TYPE "UDT_CommonStatus"
TITLE = UDT_CommonStatus
VERSION : 0.1
//User-defined structure of common statuses.
   STRUCT
      SafetyStop { ExternalAccessible := 'False'; ExternalVisible := 'False'; ExternalWritable := 'False'} : Bool;   // Emergancy stop
      Error { ExternalAccessible := 'False'; ExternalVisible := 'False'; ExternalWritable := 'False'} : Bool;   // An error is active
      Warning { ExternalAccessible := 'False'; ExternalVisible := 'False'; ExternalWritable := 'False'} : Bool;   // A warning is active
      ManualRun { ExternalAccessible := 'False'; ExternalVisible := 'False'; ExternalWritable := 'False'} : Bool;   // Running in manual mode
      Manual { ExternalAccessible := 'False'; ExternalVisible := 'False'; ExternalWritable := 'False'} : Bool;   // In manual mode
      Halted { ExternalAccessible := 'False'; ExternalVisible := 'False'; ExternalWritable := 'False'} : Bool;   // Halted
      Dieback { ExternalAccessible := 'False'; ExternalVisible := 'False'; ExternalWritable := 'False'} : Bool;   // In dieback
      Stopped { ExternalAccessible := 'False'; ExternalVisible := 'False'; ExternalWritable := 'False'} : Bool;   // Stopped
      Running { ExternalAccessible := 'False'; ExternalVisible := 'False'; ExternalWritable := 'False'} : Bool;   // Running
      EnergySave { ExternalAccessible := 'False'; ExternalVisible := 'False'; ExternalWritable := 'False'} : Bool;   // In energy saving mode
      AutoON { ExternalAccessible := 'False'; ExternalVisible := 'False'; ExternalWritable := 'False'} : Bool;   // Automatic started
   END_STRUCT;

END_TYPE

TYPE "UDT_GINStandard"
VERSION : 0.1
   STRUCT
      Destination : Array[0..20] of DInt;   // Destination
      Identification : Struct   // Barcode identification
         GoodRead { ExternalAccessible := 'False'; ExternalVisible := 'False'; ExternalWritable := 'False'} : Bool;   // Barcode read was succesful
         NoRead { ExternalAccessible := 'False'; ExternalVisible := 'False'; ExternalWritable := 'False'} : Bool;   // Barcode read was unsuccesful
         MultiRead { ExternalAccessible := 'False'; ExternalVisible := 'False'; ExternalWritable := 'False'} : Bool;   // Multiple Barcodes were detected
         Barcode : Array[0..10] of Char;   // Barcode values
      END_STRUCT;
      GinAssigned { ExternalAccessible := 'False'; ExternalVisible := 'False'; ExternalWritable := 'False'} : Bool;   // GIN is assigned to package
      Lost { ExternalAccessible := 'False'; ExternalVisible := 'False'; ExternalWritable := 'False'} : Bool;   // Lost in tracking
      Length : Int;   // Length in mm
      Width : Int;   // Width in mm
      Height : Int;   // Height in mm
      Weight : DInt;   // Weight in g
      PkgTooLong { ExternalAccessible := 'False'; ExternalVisible := 'False'; ExternalWritable := 'False'} : Bool;   // Package is too long
      PkgTooSmall { ExternalAccessible := 'False'; ExternalVisible := 'False'; ExternalWritable := 'False'} : Bool;   // Package is too small
      PkgTooHigh { ExternalAccessible := 'False'; ExternalVisible := 'False'; ExternalWritable := 'False'} : Bool;   // Package is too high
      PkgOverWeight { ExternalAccessible := 'False'; ExternalVisible := 'False'; ExternalWritable := 'False'} : Bool;   // Package is over weight
      TrailingGap : Int;   // Trailing gap size in cm between the package
      LeadingGap : Int;   // Leading gap size in cm between the package
      NrOfRecirculations : Int;   // Number of recirculations
      DestReqSend { ExternalAccessible := 'False'; ExternalVisible := 'False'; ExternalWritable := 'False'} : Bool;   // Destination request sent to high level
      DestRcv { ExternalAccessible := 'False'; ExternalVisible := 'False'; ExternalWritable := 'False'} : Bool;   // Destination received from high level
      SortStatus : Struct   // Sort status of the package
         DivertDestination : Int;   // Destination to which the package is diverted
         GoodDivert { ExternalAccessible := 'False'; ExternalVisible := 'False'; ExternalWritable := 'False'} : Bool;   // Package diverted
         FailedDivert { ExternalAccessible := 'False'; ExternalVisible := 'False'; ExternalWritable := 'False'} : Bool;   // Package failed to divert
         NoDivert : Bool := TRUE;   // Divert is not activated
         NoDivertCause : Struct   // Cause for no divert
            ChuteJam { ExternalAccessible := 'False'; ExternalVisible := 'False'; ExternalWritable := 'False'} : Bool;   // Chute is jammed
            ChuteFull { ExternalAccessible := 'False'; ExternalVisible := 'False'; ExternalWritable := 'False'} : Bool;   // Chute is full
            NoRTR { ExternalAccessible := 'False'; ExternalVisible := 'False'; ExternalWritable := 'False'} : Bool;   // Downstream conveyor is not ready to receive
            DestDisabled { ExternalAccessible := 'False'; ExternalVisible := 'False'; ExternalWritable := 'False'} : Bool;   // Destination is disabled
            TrayDisabled { ExternalAccessible := 'False'; ExternalVisible := 'False'; ExternalWritable := 'False'} : Bool;   // Tray is disabled
            SorterNotAtSpeed { ExternalAccessible := 'False'; ExternalVisible := 'False'; ExternalWritable := 'False'} : Bool;   // Sorter is not at speed
            LeadingGapError { ExternalAccessible := 'False'; ExternalVisible := 'False'; ExternalWritable := 'False'} : Bool;   // Gap size with downstream parcel is not enough
            TrailingGapError { ExternalAccessible := 'False'; ExternalVisible := 'False'; ExternalWritable := 'False'} : Bool;   // Gap size with upstream parcel is not enough
            PkgTooHigh { ExternalAccessible := 'False'; ExternalVisible := 'False'; ExternalWritable := 'False'} : Bool;   // Package is too high to divert
            PkgTooLong { ExternalAccessible := 'False'; ExternalVisible := 'False'; ExternalWritable := 'False'} : Bool;   // Package is too long to divert
            DestNotReachable { ExternalAccessible := 'False'; ExternalVisible := 'False'; ExternalWritable := 'False'} : Bool;   // Sort destionation is not reachable
            InvalidDest { ExternalAccessible := 'False'; ExternalVisible := 'False'; ExternalWritable := 'False'} : Bool;   // Sort destination is invalid
            DestTooLate { ExternalAccessible := 'False'; ExternalVisible := 'False'; ExternalWritable := 'False'} : Bool;   // Destination too late
            NoDestRcv { ExternalAccessible := 'False'; ExternalVisible := 'False'; ExternalWritable := 'False'} : Bool;   // Destination not received from high level
         END_STRUCT;
      END_STRUCT;
   END_STRUCT;

END_TYPE

TYPE "UDT_GINFedEx"
VERSION : 0.1
   STRUCT
      Timestamp : String[17];   // Local time timestamp
      TimeZoneDesignator : String[5];   // Time zone designator
      PackageEntrancePoint : String[14];   // Entrance point, where LLC starts tracking the parcel.
      PackageEntranceState : String[1];   // Entrance state
      PackageExitPoint : String[14];   // Exit point name, where LLC reports the last known tracking point.
      PackageExitState : String[1];   // Exit point state when LLC reports the last known tracking point.
      PalletType : String[2];   // Pallet code for different type of pallets on the market
      Mask : String[1];   // Flag to indicate that a pallet has been mask.
      CellNumber : String[4];   // Tray/Cell number (for loop sorters) or generated by LLC (on line sorters).
      CellsOccupied : String[1];   // Cells occupied by the piece for loop sorters.
      ImageID : String[6];   // Image ID number created by the ADC system.
      ScanUnitType : String[1];   // Scan unit type
      ADCSystemID : String[15];   // Number assigned by the ADC system
      PackageID : String[15];   // Number assigned by the LLC system
      LLCSystemID : String[15];
      HLCPackageID : String[10];   // Unique number for the specific package during it stays in HLC system.
      HLCResultCode : String[16];   // Result code based on processing of the scan event messages.
      ShipmentID : String[6];   // Consignment id of the parcel.
      WeightStatus : String[1];   // Status to indicate if the parcel/pallet has weight on the system.
      ActualDestination : String[6];   // Location code value that describes the actual disposition of the package.
      Destination1 : String[6];   // Location code value that describes where the package should go (Diverter Number).
      Destination2 : String[6];   // Location code value that describes where the package should go (Diverter Number).
      Destination3 : String[6];   // Location code value that describes where the package should go (Diverter Number).
      Destination4 : String[6];   // Location code value that describes where the package should go (Diverter Number).
      Destination5 : String[6];   // Location code value that describes where the package should go (Diverter Number).
      CutOffTimeDestination1 : String[5];   // Cut Off Time in Local Time.
      CutOffTimeDestination2 : String[5];   // Cut Off Time in Local Time.
      CutOffTimeDestination3 : String[5];   // Cut Off Time in Local Time.
      CutOffTimeDestination4 : String[5];   // Cut Off Time in Local Time.
      CutOffTimeDestination5 : String[5];   // Cut Off Time in Local Time.
      ReasonCode1 : String[8];   // Management Code value that describes the result of attempting to route the package to the Destination
      ReasonCode2 : String[8];   // Management Code value that describes the result of attempting to route the package to the Destination
      ReasonCode3 : String[8];   // Management Code value that describes the result of attempting to route the package to the Destination
      ReasonCode4 : String[8];   // Management Code value that describes the result of attempting to route the package to the Destination
      ReasonCode5 : String[8];   // Management Code value that describes the result of attempting to route the package to the Destination
      HLCDataText : String[20];   // Free text for future use.
      Customs : String[1];   // Need to be checked by customs
      DIMSystemID : String[15];   // Identifier of dimensioning system.
      DIMStatus : String[5];   // Basic diagnostic information from the dimensioning system at the moment of the measurement.
      PackageDimLength : String[6];   // Length dimension of package in resolution of dim system.
      PackageDimWidth : String[6];   // Width dimension of package in resolution of dim system.
      PackageDimHeight : String[6];   // Height dimension of package in resolution of dim system.
      DIMUOM : String[2];   // Unit of measure of the package dimensions.
      DimLFTstatusCode : String[8];   // Dimension LFT status code.
      DimConfidence : String[2];   // The level of assurance for the correct dimensions.
      DimensionSource : String[1];   // For combined camera/laser dim acquisition devices. It indicates type of capturing mode
      AlibiDims : String[25];   // Alibi for Dimensions
      SCLSystemID : String[15];   // Identifier of weight scale.
      SCLStatus : String[5];   // Basic diagnostic information from the weight scale system.
      SCLWT : String[6];   // Scale weight of package in resolution of scale system.
      SCLWTUOM : String[2];   // Unit of measurement for Weight
      SCLLFTStatusCode : String[2];   // Scale LFT status code.
      AlibiWeight : String[25];   // Alibi for Weight
      ReasonCode : String[1];   // This code should be used when the SI message has some defect.
      Stackable : String[1];   // If stackable recognition is enabled, Y or N
      Stickerstype : String[2];   // When optical recognition is used to sort
      FlyingDocument : String[1];   // Status to confirm if the document/flyer is prone to fly off the sorter.
      ModeofOperation : String[1];   // Camera Tunnel operational mode format:
      CameraHeadstatus : String[2];   // Diagnostic information on camera/laser heads performing barcode reads.
      PackageDataTruncated : String[1];   // Y = Full length of barcode data exceeds 9999 bytes, data truncated
      TotalBarcodeDataLength : String[4];   // Length of all barcode data that was sent in bytes;
      Barcode1Identification : String[3];   // Barcode identifier code.
      Barcode1status : String[2];   // Barcode confidence factor
      Barcode1datalength : String[4];   // String length of barcode data in bytes; inclusive of this field. Use 0054 as a fixed value
      Barcode1data : String[50];   // Highest priority barcode
      Barcode2Identification : String[3];   // Barcode identifier code.
      Barcode2status : String[2];   // Barcode confidence factor
      Barcode2datalength : String[4];   // String length of barcode data in bytes; inclusive of this field. Use 0054 as a fixed value
      Barcode2data : String[50];   // Highest priority barcode
      Barcode3Identification : String[3];   // Barcode identifier code.
      Barcode3status : String[2];   // Barcode confidence factor
      Barcode3datalength : String[4];   // String length of barcode data in bytes; inclusive of this field. Use 0054 as a fixed value
      Barcode3data : String[50];   // Highest priority barcode
      BarcodeIdentification : String[3];   // Barcode identifier code.
      Barcodestatus : String[2];   // Barcode confidence factor
      Barcodedatalength : String[4];   // String length of barcode data in bytes
      Barcodedata : String[50];   // Sortation barcode
      CustomerID : DInt;   // 6 digits SequentialID (NNNNNN)
      AreaNumber : String[2];   // Package Sequence ID "Area Number"
      PurgeEnabled { ExternalAccessible := 'False'; ExternalVisible := 'False'; ExternalWritable := 'False'} : Bool;   // Purge enabled for parcel: destination overwritten with Purge destination
   END_STRUCT;

END_TYPE

TYPE "UDT_GINUPS"
VERSION : 0.1
   STRUCT
      TRKNUM : String[18];   // Tracking number
      PKGUID : String[32];   // Package ID
      MSGID : String[32];   // Message ID
      Length : Int;   // Camera Length in mm
      Width : Int;   // Camera Width in mm
      Height : Int;   // Camera Height in mm
      Weight : DInt;   // Weight in g
      IDCreated { ExternalAccessible := 'False'; ExternalVisible := 'False'; ExternalWritable := 'False'} : Bool;   // Byte 1, Bit 0 - PLCID created or TrayID Read
      DimDataRcv { ExternalAccessible := 'False'; ExternalVisible := 'False'; ExternalWritable := 'False'} : Bool;   // Byte 1, Bit 1 - Package Dimensional Data Received via Camera Scan Data Message
      PkgWrongInduct { ExternalAccessible := 'False'; ExternalVisible := 'False'; ExternalWritable := 'False'} : Bool;   // Byte 1, Bit 2 - Package Did NOT Induct Properly (Non-Tray Systems)
      IDCalcFromCamID { ExternalAccessible := 'False'; ExternalVisible := 'False'; ExternalWritable := 'False'} : Bool;   // Byte 2, Bit 0 - PLCID/TrayID Calculated From CamID
      UnknownParcelID { ExternalAccessible := 'False'; ExternalVisible := 'False'; ExternalWritable := 'False'} : Bool;   // Byte 2, Bit 4 - Unknown Parcel ID
      UndefinedProblem { ExternalAccessible := 'False'; ExternalVisible := 'False'; ExternalWritable := 'False'} : Bool;   // Byte 2, Bit 5 - Un-Defined Problem
      UnrecognizedCmd { ExternalAccessible := 'False'; ExternalVisible := 'False'; ExternalWritable := 'False'} : Bool;   // Byte 2, Bit 6 - Un-recognized command
      SorterInMainteneceMode { ExternalAccessible := 'False'; ExternalVisible := 'False'; ExternalWritable := 'False'} : Bool;   // Byte 2, Bit 7 - Sorter in Maintenance/Commissioning Mode
      DestUserSusp { ExternalAccessible := 'False'; ExternalVisible := 'False'; ExternalWritable := 'False'} : Bool;   // Byte 3, Bit 3 - Destination User Suspended
      SorterNotSynch { ExternalAccessible := 'False'; ExternalVisible := 'False'; ExternalWritable := 'False'} : Bool;   // Byte 3, Bit 6 - Sorter NOT Synchronized (Tilt Tray Systems)
      PkgDetAtVerCheckPoint { ExternalAccessible := 'False'; ExternalVisible := 'False'; ExternalWritable := 'False'} : Bool;   // Byte 4, Bit 0 - Package Detected at Verification Check Point
      ChuteFullAftrAlterDest { ExternalAccessible := 'False'; ExternalVisible := 'False'; ExternalWritable := 'False'} : Bool;   // Byte 4, Bit 7 - Preferred chute full after passed alternate destination
      ChuteNotAvailAfterAlterDest { ExternalAccessible := 'False'; ExternalVisible := 'False'; ExternalWritable := 'False'} : Bool;   // Byte 5, Bit 0 - Preferred chute not available after passed alternate destination
      PLCRedirected { ExternalAccessible := 'False'; ExternalVisible := 'False'; ExternalWritable := 'False'} : Bool;   // Byte 5, Bit 2 - PLC Redirected
      ThreatParcel { ExternalAccessible := 'False'; ExternalVisible := 'False'; ExternalWritable := 'False'} : Bool;   // Threat parcel
   END_STRUCT;

END_TYPE

TYPE "UDT_GINDHL"
VERSION : 0.1
   STRUCT
      ObjectID : String[10];   // Object ID
      VID : String[16];   // Virtual Item Identifier (VID)
      PieceID : String[40];   // Piece ID barcodes
      SortStrategy : String[1];   // Sort Strategy 1 - Highest priority available , 2 - Nearest
      ParcelReject { ExternalAccessible := 'False'; ExternalVisible := 'False'; ExternalWritable := 'False'} : Bool;   // True - Parcel reject
      Destination : Array[1..6] of Struct   // Destination
         ID : UInt;   // ID
         SortCommandActive { ExternalAccessible := 'False'; ExternalVisible := 'False'; ExternalWritable := 'False'} : Bool;   // Sort command
         ParcelSorted { ExternalAccessible := 'False'; ExternalVisible := 'False'; ExternalWritable := 'False'} : Bool;   // Parcel sorted
         Rejected { ExternalAccessible := 'False'; ExternalVisible := 'False'; ExternalWritable := 'False'} : Bool;   // Parcel rejected
         Reason : Int;   // Reason
      END_STRUCT;
      ParcelLocation : Struct   // Parcel Location
         Current : UInt;   // Current
         Last : UInt;   // Last
         Sort : UInt;   // Sort
      END_STRUCT;
      MFCMessage : Struct   // MFC Sort messages
         Sent : Struct   // Messages sent from the PLC to the MFC system
            SortResult { ExternalAccessible := 'False'; ExternalVisible := 'False'; ExternalWritable := 'False'} : Bool;   // Message Sort Result
            VIDResponse { ExternalAccessible := 'False'; ExternalVisible := 'False'; ExternalWritable := 'False'} : Bool;   // Message VID Response
            ScanReset { ExternalAccessible := 'False'; ExternalVisible := 'False'; ExternalWritable := 'False'} : Bool;   // Message Scan Reset
            XrayResult { ExternalAccessible := 'False'; ExternalVisible := 'False'; ExternalWritable := 'False'} : Bool;   // Message Xray result
            ParcelRegInfo { ExternalAccessible := 'False'; ExternalVisible := 'False'; ExternalWritable := 'False'} : Bool;   // Message Xray registration info
         END_STRUCT;
         Received : Struct   // Messages received from the MFC system to the PLC
            RejectParcel { ExternalAccessible := 'False'; ExternalVisible := 'False'; ExternalWritable := 'False'} : Bool;   // Message Reject Parcel
            Destination { ExternalAccessible := 'False'; ExternalVisible := 'False'; ExternalWritable := 'False'} : Bool;   // Message Destination
            DestinationResent { ExternalAccessible := 'False'; ExternalVisible := 'False'; ExternalWritable := 'False'} : Bool;   // Message Destination Resent
            TemporaryParcelIdentifier { ExternalAccessible := 'False'; ExternalVisible := 'False'; ExternalWritable := 'False'} : Bool;   // Message Temporary Parcel Identifier
            XrayRegistrationInfo { ExternalAccessible := 'False'; ExternalVisible := 'False'; ExternalWritable := 'False'} : Bool;
         END_STRUCT;
      END_STRUCT;
      Xray : Struct   // Xray data structure
         RoutingCode : String[2];   // Routing code
         Group : String[1];   // The group field is used to identify the group of the operator decisions came from in a
         Level : String[1];   // Level field is used to identify which level the operator decision came from in a
         Result : String[1];   // Results can be indicated with the following:A = Accept, R = Reject, U = Unavailable (Timeout), Z = High Threat
         BagIDMessage : Struct   // Message from PLC to Xray
            MessagePrepared { ExternalAccessible := 'False'; ExternalVisible := 'False'; ExternalWritable := 'False'} : Bool;   // The message is prepared and ready to send
            WrongMessageStructure { ExternalAccessible := 'False'; ExternalVisible := 'False'; ExternalWritable := 'False'} : Bool;   // The message has wrong structure
            Sent { ExternalAccessible := 'False'; ExternalVisible := 'False'; ExternalWritable := 'False'} : Bool;   // The message sent by PLC to Xray
            SentTime : String;   // Time when message sent by PLC to Xray
            NotSent { ExternalAccessible := 'False'; ExternalVisible := 'False'; ExternalWritable := 'False'} : Bool;   // The message was not sent from the PLC
            Received { ExternalAccessible := 'False'; ExternalVisible := 'False'; ExternalWritable := 'False'} : Bool;   // The message received by Xray
            TimeReceived : String;   // Time when message received by Xray
            NotReceived { ExternalAccessible := 'False'; ExternalVisible := 'False'; ExternalWritable := 'False'} : Bool;   // The message did not reach Xray
         END_STRUCT;
         DecisionMessage : Struct   // Message from Xray to PLC
            Received { ExternalAccessible := 'False'; ExternalVisible := 'False'; ExternalWritable := 'False'} : Bool;   // The message received by PLC
            ReceivedTime : String;   // The message received by PLC
            NotReceivedOnTime { ExternalAccessible := 'False'; ExternalVisible := 'False'; ExternalWritable := 'False'} : Bool;   // The message did not reach PLC
         END_STRUCT;
      END_STRUCT;
   END_STRUCT;

END_TYPE

TYPE "UDT_GINWCS"
VERSION : 0.1
   STRUCT
      ActionTaken : String;   // Location code value that describes the actual disposition of the package
      Destination1 : String[20];   // Location code value that describes where the package should go (Diverter Number)
      Destination2 : String[20];   // Location code value that describes where the package should go (Diverter Number)
      Destination3 : String[20];   // Location code value that describes where the package should go (Diverter Number)
      Destination4 : String[20];   // Location code value that describes where the package should go (Diverter Number)
      Destination5 : String[20];   // Location code value that describes where the package should go (Diverter Number)
      ReasonCode : String[2];   // Management Code value that describes the result of attempting to route the package to the Destination
      Barcode1 : String;   // Barcode identifier code
      Barcode2 : String;
      Barcode3 : String;
      Barcode4 : String;
   END_STRUCT;

END_TYPE

TYPE "UDT_GINWES"
VERSION : 0.1
   STRUCT
      Barcode : String[40];
   END_STRUCT;

END_TYPE

TYPE "UDT_UPSHealth"
TITLE = UDT_Health
VERSION : 0.1
//User-defined structure of UPS health message data.
   STRUCT
      "Type" : String;
      Failure : DInt;
      Model : String;
      Error : Bool;
   END_STRUCT;

END_TYPE

TYPE "UDT_FifoStatus"
TITLE = UDT_FifoStatus
VERSION : 0.1
//
//User-defined structure of FC_Fifo function status.
//Version History:
//Date              | Version   | Author         | Remark
//24/05/2019  | 0.1           | K.Pokorski   | first release MHSE TIA 15.1
//24/05/2019  | 0.2           | K.Pokorski   | first release MHSE TIA 15.1
//
   STRUCT
      InvalidMode { ExternalAccessible := 'False'; ExternalVisible := 'False'; ExternalWritable := 'False'} : Bool;   // Invalid mode selected
      InvalidMaxNrOfEntries { ExternalAccessible := 'False'; ExternalVisible := 'False'; ExternalWritable := 'False'} : Bool;   // Invalid maximum number of entries or buffer is not an array
      InvalidTotalEntriesStored { ExternalAccessible := 'False'; ExternalVisible := 'False'; ExternalWritable := 'False'} : Bool;   // Invalid total number of entries
      InvalidNextEntryToWrite { ExternalAccessible := 'False'; ExternalVisible := 'False'; ExternalWritable := 'False'} : Bool;   // Invalid number of next entry to write
      InvalidNextEntryToRead { ExternalAccessible := 'False'; ExternalVisible := 'False'; ExternalWritable := 'False'} : Bool;   // Invalid number of next entry to read
      InvalidDataType { ExternalAccessible := 'False'; ExternalVisible := 'False'; ExternalWritable := 'False'} : Bool;   // Message and buffer element data type inconsistent
      FifoPreFull { ExternalAccessible := 'False'; ExternalVisible := 'False'; ExternalWritable := 'False'} : Bool;   // 90 % of FIFO data buffer capacity reached
      FifoFull { ExternalAccessible := 'False'; ExternalVisible := 'False'; ExternalWritable := 'False'} : Bool;   // FIFO data buffer full
   END_STRUCT;

END_TYPE

DATA_BLOCK "DB_Memory"
TITLE = DB_Memory
{ S7_Optimized_Access := 'TRUE' }
AUTHOR : MHSE
VERSION : 3.0
NON_RETAIN
   VAR
      ClockByte { ExternalAccessible := 'False'; ExternalVisible := 'False'; ExternalWritable := 'False'} : Byte;   // System clock byte
      Clock_10Hz { ExternalAccessible := 'False'; ExternalVisible := 'False'; ExternalWritable := 'False'} : Bool;   // 10 Hz system clock bit
      Clock_5Hz { ExternalAccessible := 'False'; ExternalVisible := 'False'; ExternalWritable := 'False'} : Bool;   // 5 Hz system clock bit
      "Clock_2.5Hz" { ExternalAccessible := 'False'; ExternalVisible := 'False'; ExternalWritable := 'False'} : Bool;   // 2.5 Hz system clock bit
      Clock_2Hz { ExternalAccessible := 'False'; ExternalVisible := 'False'; ExternalWritable := 'False'} : Bool;   // 2 Hz system clock bit
      "Clock_1.25Hz" { ExternalAccessible := 'False'; ExternalVisible := 'False'; ExternalWritable := 'False'} : Bool;   // 1.25 Hz system clock bit
      Clock_1Hz { ExternalAccessible := 'False'; ExternalVisible := 'False'; ExternalWritable := 'False'} : Bool;   // 1 Hz system clock bit
      "Clock_0.625Hz" { ExternalAccessible := 'False'; ExternalVisible := 'False'; ExternalWritable := 'False'} : Bool;   // 0.625 Hz system clock bit
      "Clock_0.5Hz" { ExternalAccessible := 'False'; ExternalVisible := 'False'; ExternalWritable := 'False'} : Bool;   // 0.5 Hz system clock bit
      SystemByte { ExternalAccessible := 'False'; ExternalVisible := 'False'; ExternalWritable := 'False'} : Byte;   // System byte
      OSClockByte { ExternalAccessible := 'False'; ExternalVisible := 'False'; ExternalWritable := 'False'} : Byte;   // One shot of clock pulse
      "OS_0.1sec" { ExternalAccessible := 'False'; ExternalVisible := 'False'; ExternalWritable := 'False'} : Bool;   // One shot every 0.1 sec
      "OS_0.2sec" { ExternalAccessible := 'False'; ExternalVisible := 'False'; ExternalWritable := 'False'} : Bool;   // One shot every 0.2 sec
      "OS_0.4sec" { ExternalAccessible := 'False'; ExternalVisible := 'False'; ExternalWritable := 'False'} : Bool;   // One shot every 0.4 sec
      "OS_0.5sec" { ExternalAccessible := 'False'; ExternalVisible := 'False'; ExternalWritable := 'False'} : Bool;   // One shot every 0.5 sec
      "OS_0.8sec" { ExternalAccessible := 'False'; ExternalVisible := 'False'; ExternalWritable := 'False'} : Bool;   // One shot every 0.8 sec
      OS_1sec { ExternalAccessible := 'False'; ExternalVisible := 'False'; ExternalWritable := 'False'} : Bool;   // One shot every 1 sec
      "OS_1.6sec" { ExternalAccessible := 'False'; ExternalVisible := 'False'; ExternalWritable := 'False'} : Bool;   // One shot every 1.6 sec
      OS_2sec { ExternalAccessible := 'False'; ExternalVisible := 'False'; ExternalWritable := 'False'} : Bool;   // One shot every 2 sec
      PrevCycleTime { ExternalAccessible := 'False'; ExternalVisible := 'False'; ExternalWritable := 'False'} : LReal;   // Previous PLC cycle Time
      RuntimeMem { ExternalAccessible := 'False'; ExternalVisible := 'False'; ExternalWritable := 'False'} : LReal;   // Runtime memory
      FirstScan { ExternalAccessible := 'False'; ExternalVisible := 'False'; ExternalWritable := 'False'} : Bool;   // First scan bit
      DiagStatusUpdate { ExternalAccessible := 'False'; ExternalVisible := 'False'; ExternalWritable := 'False'} : Bool;   // Diagnostic status update
      AlwaysTrue { ExternalAccessible := 'False'; ExternalVisible := 'False'; ExternalWritable := 'False'} : Bool;   // Always True bit
      AlwaysFalse { ExternalAccessible := 'False'; ExternalVisible := 'False'; ExternalWritable := 'False'} : Bool;   // Always False bit
      CommissioningFalse { ExternalAccessible := 'False'; ExternalVisible := 'False'; ExternalWritable := 'False'} : Bool;   // Commissioning always false
      CommissioningTrue { ExternalAccessible := 'False'; ExternalVisible := 'False'; ExternalWritable := 'False'} : Bool;   // Commissioning always true
      ReconnectCommand { ExternalAccessible := 'False'; ExternalVisible := 'False'; ExternalWritable := 'False'} : Bool;   // Reconnect command
      ScanMainRack { ExternalAccessible := 'False'; ExternalVisible := 'False'; ExternalWritable := 'False'} : Bool;   // Trigger to check main rack confiuration
      ScanProfinet { ExternalAccessible := 'False'; ExternalVisible := 'False'; ExternalWritable := 'False'} : Bool;   // Scan profinet bit
      Simulation { ExternalAccessible := 'False'; ExternalVisible := 'False'; ExternalWritable := 'False'} : Bool;   // Simulation
      PN1OK { ExternalAccessible := 'False'; ExternalVisible := 'False'; ExternalWritable := 'False'} : Bool;   // Profinet ok
      "Local~PROFINET_IO-System" { ExternalAccessible := 'False'; ExternalVisible := 'False'; ExternalWritable := 'False'} : HW_ANY;   // HW Intentifier of PN-IO System
      "Local~PROFINET_IO-System_1" { ExternalAccessible := 'False'; ExternalVisible := 'False'; ExternalWritable := 'False'} : HW_ANY;   // HW Intentifier of PN-IOSystem 1
      "Local~PROFINET_IO-System_2" { ExternalAccessible := 'False'; ExternalVisible := 'False'; ExternalWritable := 'False'} : HW_ANY;   // HW Intentifier of PN-IOSystem 2
      "Local~PROFINET_IO-System_3" { ExternalAccessible := 'False'; ExternalVisible := 'False'; ExternalWritable := 'False'} : HW_ANY;   // HW Intentifier of PN-IOSystem 3
      "Local~PROFINET_IO-System_4" { ExternalAccessible := 'False'; ExternalVisible := 'False'; ExternalWritable := 'False'} : HW_ANY;   // HW Intentifier of PN-IOSystem 4
      "Local~PROFINET_IO-System_5" { ExternalAccessible := 'False'; ExternalVisible := 'False'; ExternalWritable := 'False'} : HW_ANY;   // HW Intentifier of PN-IOSystem 5
      "Local~PROFINET_IO-System_6" { ExternalAccessible := 'False'; ExternalVisible := 'False'; ExternalWritable := 'False'} : HW_ANY;   // HW Intentifier of PN-IOSystem 6
      "Local~PROFINET_IO-System_7" { ExternalAccessible := 'False'; ExternalVisible := 'False'; ExternalWritable := 'False'} : HW_ANY;   // HW Intentifier of PN-IOSystem 7
      "Local~PROFINET_IO-System_8" { ExternalAccessible := 'False'; ExternalVisible := 'False'; ExternalWritable := 'False'} : HW_ANY;   // HW Intentifier of PN-IOSystem 8
      "Local~PROFINET_IO-System_9" { ExternalAccessible := 'False'; ExternalVisible := 'False'; ExternalWritable := 'False'} : HW_ANY;   // HW Intentifier of PN-IOSystem 9
   END_VAR


BEGIN

END_DATA_BLOCK

TYPE "UDT_GIN"
VERSION : 0.1
   STRUCT
      General { S7_SetPoint := 'False'} : "UDT_GINStandard";
      FedEx { S7_SetPoint := 'False'} : "UDT_GINFedEx";
      UPS { S7_SetPoint := 'False'} : "UDT_GINUPS";
      DHL { S7_SetPoint := 'False'} : "UDT_GINDHL";
      WCS { S7_SetPoint := 'False'} : "UDT_GINWCS";
      WES { S7_SetPoint := 'False'} : "UDT_GINWES";
   END_STRUCT;

END_TYPE

TYPE "UDT_FifoHeader"
TITLE = UDT_FifoHeader
VERSION : 0.1
//User-defined structure of FIFO register header information.
   STRUCT
      Status : Struct   // Status bits
         Empty { ExternalAccessible := 'False'; ExternalVisible := 'False'; ExternalWritable := 'False'} : Bool;   // FIFO Empty
         Prefull { ExternalAccessible := 'False'; ExternalVisible := 'False'; ExternalWritable := 'False'} : Bool;   // FIFO Prefull
         Full { ExternalAccessible := 'False'; ExternalVisible := 'False'; ExternalWritable := 'False'} : Bool;   // FIFO Full
      END_STRUCT;
      NextEntryToRead : Int;   // Next FIFO entry to read
      NextEntryToWrite : Int;   // Next FIFO entry to write
      MaxNrOfEntries : Int;   // Maximum number of FIFO entries
      TotalEntriesStored : Int;   // Total number of FIFO entries
   END_STRUCT;

END_TYPE

TYPE "UDT_EventStatistic"
TITLE = UDT_EventStatistic
VERSION : 0.1
//User-defined structure of event statistic data.
   STRUCT
      NumberOfTimes : DInt;   // Number of times the event occurred since last reset
      LastEventSeconds : DInt;   // Number of seconds of the current or last event
      TotalEventSeconds : DInt;   // Total number of seconds the event occurred since last reset
   END_STRUCT;

END_TYPE

TYPE "UDT_EquipmentControl"
TITLE = UDT_EquipmentControl
VERSION : 0.1
//User-defined structure of equipment control commands.
   STRUCT
      Command : Struct   // Control command
         Start { ExternalAccessible := 'False'; ExternalVisible := 'False'; ExternalWritable := 'False'} : Bool;   // Start conveyor
         Stop { ExternalAccessible := 'False'; ExternalVisible := 'False'; ExternalWritable := 'False'} : Bool;   // Stop conveyor
         Reset { ExternalAccessible := 'False'; ExternalVisible := 'False'; ExternalWritable := 'False'} : Bool;   // Faults reset
         ResetData { ExternalAccessible := 'False'; ExternalVisible := 'False'; ExternalWritable := 'False'} : Bool;   // Statistics reset
         ManualMode { ExternalAccessible := 'False'; ExternalVisible := 'False'; ExternalWritable := 'False'} : Bool;   // Manual mode required
         DisableManualMode { ExternalAccessible := 'False'; ExternalVisible := 'False'; ExternalWritable := 'False'} : Bool;   // Disable manual mode
         AutomaticOn { ExternalAccessible := 'False'; ExternalVisible := 'False'; ExternalWritable := 'False'} : Bool;   // System is started in automatic mode
         StopRequest { ExternalAccessible := 'False'; ExternalVisible := 'False'; ExternalWritable := 'False'} : Bool;
      END_STRUCT;
      Report { S7_SetPoint := 'False'} : "UDT_CommonStatus";   // Conveyors state
      Request : Struct   // Request from equipment
         RestartRequired { ExternalAccessible := 'False'; ExternalVisible := 'False'; ExternalWritable := 'False'} : Bool;   // Restart required from system control
         SignalingRequest { ExternalAccessible := 'False'; ExternalVisible := 'False'; ExternalWritable := 'False'} : Bool;   // Beeper required
         InhibitStop { ExternalAccessible := 'False'; ExternalVisible := 'False'; ExternalWritable := 'False'} : Bool;
      END_STRUCT;
   END_STRUCT;

END_TYPE

FUNCTION "FC_GetNrOfArrayEl" : Int
TITLE = FC_GetNrOfArrayEl
{ S7_Optimized_Access := 'TRUE' }
AUTHOR : MHSE
FAMILY : GeneralSystemFunctions
VERSION : 3.0
// ATTRIBUTES
// AUTO_NUMBER = True
// BLOCK_NUMBER = 19
// END_ATTRIBUTES
//Function to get the number of array elements.
   VAR_INPUT
      iv_Array : Variant;   // Input array
   END_VAR

   VAR_TEMP
      ti_NrOfArrayEl : Int;   // Number of array elements
   END_VAR


BEGIN
	(*
	----------------------------------------------------------------------------------------

	Version history:
	Date        | Version   | Author        | Remark
	----------------------------------------------------------------------------------------
	24/05/2019  | 0.1       | L.Klar        | first release MHS TIA 15.1
	24/07/2019  | 2.0       | L.Klar        | 2.0 MHS library release TIA 15.1
	27/08/2019  | 2.1       | K.Pokorski    | Comments adjusted
	12/11/2019  | 3.0       | P.Majka       | 3.0 MHS library release TIA 15.1
	21/02/2023  | 4.0       | F.Baten       | 4.0 Release TIA 17.5
	*)

	REGION 1 – Number of an array elements

	    IF IS_ARRAY(#iv_Array)                                                  // Input variable is an array
	    THEN

	        #ti_NrOfArrayEl := UDINT_TO_INT(CountOfElements(#iv_Array));

	        // Reset array length if the input variable isn't an array
	    ELSE

	        #ti_NrOfArrayEl := 0;

	    END_IF;

	END_REGION

	REGION 2 – Return output

	    #FC_GetNrOfArrayEl := #ti_NrOfArrayEl;

	END_REGION

END_FUNCTION

TYPE "UDT_UPSScanData2"
TITLE = UDT_ScanData2
VERSION : 0.1
//User-defined structure of UPS SCAN_DATA2 data.
   STRUCT
      MSGID : String;
      CONFLICT_CODE : String;
      BARCODE_ZIP : String;
      BARCODE_TRACK : String;
      BARCODE_PTN : String;
      MAXI_ZIPCODE : String;
      MAXI_COUNTRY : String;
      MAXI_SERVICE : String;
      MAXI_TRACK : String;
      MAXI_SHIPPER : String;
      LENGTH1 : String;
      LENGTH2 : String;
      HEIGHT : String;
      VERTEX : String;
      ORIENTATION : String;
      OVERHANG : String;
      WEIGHT : String;
      APPENDED_DATA : Struct
         Constant_1 : String := '1';
         FRAME_ID : String;
         DIMENSION : String;
         PACKAGE_NUMBER : String;
         BARCODE_1 : String;
         DESCRIPTION_1 : String;
         BARCODE_2 : String;
         DESCRIPTION_2 : String;
         BARCODE_3 : String;
         DESCRIPTION_3 : String;
         Constant_4 : String := '4';
         SCALE_WEIGHT : String;
         Constant_5 : String := '5';
         GIRTH : String;
         Constant_6 : String := '6';
         ERROR_CODE : String;
      END_STRUCT;
   END_STRUCT;

END_TYPE

DATA_BLOCK "DB_GIN"
TITLE = DB_GIN
{ S7_Optimized_Access := 'TRUE' }
AUTHOR : MHSE
FAMILY : GeneralSystemFunctions
VERSION : 3.0
NON_RETAIN
//Data block to store parcels informations.
   VAR
      GIN { ExternalAccessible := 'False'; ExternalVisible := 'False'; ExternalWritable := 'False'; S7_SetPoint := 'False'} : Array[1..1] of "UDT_GIN";   // GIN informations - for project remove unneeded customers and extend array bound range to 9999
   END_VAR


BEGIN

END_DATA_BLOCK

TYPE "UDT_UPSMessage"
VERSION : 0.1
   STRUCT
      SCN { ExternalAccessible := 'False'; ExternalVisible := 'False'; ExternalWritable := 'False'} : String[15];   // Sender Client Name
      SCT { ExternalAccessible := 'False'; ExternalVisible := 'False'; ExternalWritable := 'False'} : String[8];   // Sender Client Type
      RCN { ExternalAccessible := 'False'; ExternalVisible := 'False'; ExternalWritable := 'False'} : String[15];   // Receiver Client Name
      RCT { ExternalAccessible := 'False'; ExternalVisible := 'False'; ExternalWritable := 'False'} : String[8];   // Receiver Client Type
      MT { ExternalAccessible := 'False'; ExternalVisible := 'False'; ExternalWritable := 'False'} : String;   // Message type
      Data { ExternalAccessible := 'False'; ExternalVisible := 'False'; ExternalWritable := 'False'} : Array[1..35] of String[32];   // Buffer for message data fields
   END_STRUCT;

END_TYPE

TYPE "UDT_UPSExternalReader"
VERSION : 0.1
   STRUCT
      NameIdentifier : String := 'CAMERA';   // Device name idetifier
      IPAddress : String[15];
      State : Bool;
      HealthMessage { S7_SetPoint := 'False'} : "UDT_UPSHealth";   // Health message data
      ScanData2Message { S7_SetPoint := 'False'} : "UDT_UPSScanData2";   // ScanData2 message data
   END_STRUCT;

END_TYPE

TYPE "UDT_Connection"
TITLE = UDT_Connection
VERSION : 0.1
//User-defined structure of connection parameters.
   STRUCT
      ActiveEstablished : Bool := FALSE;   // 0 – Passive connection establishment; 1 – Active connection establishment
      Interface_ID : HW_ANY := 64;   // Interface ID of CPU Ethernet interface
      ID : CONN_OUC;   // Unique ID as system reference for the connection
      IP : Array[1..4] of Int;   // IP address
      Port : UInt;   // Port number of the communication partner
      ConTimeout : DInt;   // Maximum waiting time for response from the communication partner [ms]
   END_STRUCT;

END_TYPE

TYPE "UDT_Message"
TITLE = UDT_Message
VERSION : 0.1
//User-defined structure of the message characters array.
   STRUCT
      Character : Array[0..499] of Char;   // Message character
   END_STRUCT;

END_TYPE

TYPE "UDT_TCPIPConnectStatistics"
TITLE = UDT_TCPIPConnectStatistics
VERSION : 0.1
//User-defined structure of FB_TCPIPConnect function block statistics.
   STRUCT
      ConnectionLost { S7_SetPoint := 'False'} : "UDT_EventStatistic";   // Connection lost statistics
   END_STRUCT;

END_TYPE

DATA_BLOCK "DB_HMIStatusConfiguration"
TITLE = DB_HMIStatusConfiguration
{ S7_Optimized_Access := 'TRUE' }
AUTHOR : MHSE
VERSION : 3.0
NON_RETAIN
   VAR
      FireAlarm : Int;   // Fire alarm active
      SafetyStop : Int;   // Safety stop error status
      Error : Int;   // Error status
      Warning : Int;   // Warning status
      ManualRun : Int;   // Manual run status
      Manual : Int;   // Manual status
      Halted : Int;   // Halted status
      Dieback : Int;   // Die back status
      Stopped : Int;   // Stopped status
      Running : Int;   // Running status
      EnergySave : Int;   // Energy save status
      CommunicationError : Int;   // Communication error status
      CBError : Int;   // CB error status
      ProfinetError : Int;   // Profinet error status
      HardwareError : Int;   // Hardware error status
      VFDNotHealthy : Int;   // VFD noth healthy status
      VFDError : Int;   // VFD error status
      PECJam : Int;   // PEC jam status
      ChuteFull : Int;   // Chute full status
      EncoderError : Int;   // Encoder error status
      TrackingError : Int;   // Tracking error status
      DimensionError : Int;   // Dimension error status
      OperationalError : Int;   // Operational error status
      AutoON : Int;   // Automatic is on
      ChuteHalfFull : Int;   // Disable by operator
      DisableByManagement : Int;   // Disable by management
      GateOpen : Int;   // Manual operated gate is open
      GateClosed : Int;   // Manual operated gate is closed
      GateClosedAndNoOperatorPresent : Int;   // Manual operated gate is closed and no operator is present
      PositionChangeOngoing : Int;   // Lifting device or arm diverter changing position
      BufferMode : Int;   // BufferMode Active
      ContinuousMode : Int;   // ContinuousMode Active
      LabbelingMode : Int;   // LabbelingMode Active
   END_VAR


BEGIN
   FireAlarm := 1;
   SafetyStop := 3;
   Error := 5;
   Warning := 7;
   ManualRun := 9;
   Manual := 11;
   Halted := 13;
   Dieback := 15;
   Stopped := 17;
   Running := 19;
   EnergySave := 21;
   CommunicationError := 23;
   CBError := 25;
   ProfinetError := 27;
   HardwareError := 29;
   VFDNotHealthy := 31;
   VFDError := 33;
   PECJam := 35;
   ChuteFull := 37;
   EncoderError := 39;
   TrackingError := 41;
   DimensionError := 43;
   OperationalError := 45;
   AutoON := 47;
   ChuteHalfFull := 49;
   DisableByManagement := 51;
   GateOpen := 53;
   GateClosed := 55;
   GateClosedAndNoOperatorPresent := 57;
   PositionChangeOngoing := 59;
   BufferMode := 61;
   ContinuousMode := 63;
   LabbelingMode := 65;

END_DATA_BLOCK

FUNCTION "FC_EquipmentReport" : Void
TITLE = FC_Equipment_Report
{ S7_Optimized_Access := 'TRUE' }
AUTHOR : MHSE
FAMILY : GeneralSystemFunctions
VERSION : 3.0
// ATTRIBUTES
// AUTO_NUMBER = True
// BLOCK_NUMBER = 16
// END_ATTRIBUTES
//Function to generate equipment report.
   VAR_INPUT
      iUDT_Status : "UDT_CommonStatus";   // Status structure
   END_VAR

   VAR_IN_OUT
      iqUDT_Control : "UDT_EquipmentControl";   // Equipment control
   END_VAR


BEGIN
	(*
	----------------------------------------------------------------------------------------

	Version history:
	Date        | Version   | Author        | Remark
	----------------------------------------------------------------------------------------
	24/05/2019  | 0.1       | F.Baten       | first release MHS TIA 15.1
	17/06/2019  | 0.3       | L.Klar        | Manual mode added to "UDT_EquipmentControl"
	17/07/2019  | 0.4       | A.Nowak       | Add all statuses and comments
	24/07/2019  | 2.0       | L.Klar        | 2.0 MHS library release TIA 15.1
	27/08/2019  | 2.1       | K.Pokorski    | Comments adjusted
	16/09/2019  | 2.2       | K.Pokorski    | Equipment error free condition added to "Restart required" status
	06/10/2019  | 2.3       | S. Deukar     | Updated accoring to new UDT equipment report
	12/11/2019  | 3.0       | P.Majka       | 3.0 MHS library release TIA 15.1
	05/02/2024  | 3.1       | L.Klar        | Auto On extention added
	13/03/2024  | 4.0       | S. Nieswiec   | Added to baseline
	*)

	REGION 1 - Equipment report update

	    // Extension of stopped equipment report with the stopped status
	    #iqUDT_Control.Report.Stopped := #iUDT_Status.Stopped
	    OR #iqUDT_Control.Report.Stopped;

	    // Extension of started equipment report with the started status
	    #iqUDT_Control.Report.Running := #iUDT_Status.Running
	    OR #iqUDT_Control.Report.Running;

	    // Extension of energy save equipment report with the energy save status
	    #iqUDT_Control.Report.EnergySave := #iUDT_Status.EnergySave
	    OR #iqUDT_Control.Report.EnergySave;

	    // Extension of warning equipment report with the warning status
	    #iqUDT_Control.Report.Warning := #iUDT_Status.Warning
	    OR #iqUDT_Control.Report.Warning;

	    // Extension of manual mode equipment report with the manual mode status
	    #iqUDT_Control.Report.Manual := #iUDT_Status.Manual
	    OR #iqUDT_Control.Report.Manual;

	    // Extension of error equipment report with the error status
	    #iqUDT_Control.Report.Error := #iUDT_Status.Error
	    OR #iqUDT_Control.Report.Error;

	    // Extension of safety stop equipment report with the safety stop status
	    #iqUDT_Control.Report.SafetyStop := #iUDT_Status.SafetyStop
	    OR #iqUDT_Control.Report.SafetyStop;

	    // Extension of Auto On equipment report with the Auto On status
	    #iqUDT_Control.Report.AutoON := #iUDT_Status.AutoON
	    OR #iqUDT_Control.Report.AutoON;

	    // Extension of restart required equipment report with the restart required and no equipment error statuses
	    #iqUDT_Control.Request.RestartRequired := #iUDT_Status.Stopped
	    AND NOT #iUDT_Status.Error
	    OR #iqUDT_Control.Request.RestartRequired;

	END_REGION
END_FUNCTION

FUNCTION "FC_Statistics" : Void
TITLE = FC_Statistics
{ S7_Optimized_Access := 'TRUE' }
AUTHOR : MHSE
FAMILY : GeneralSystemFunctions
VERSION : 3.0
// ATTRIBUTES
// AUTO_NUMBER = True
// BLOCK_NUMBER = 26
// END_ATTRIBUTES
//Function to calculate statistics.
   VAR_INPUT
      ix_Reset : Bool;   // Reset statistics data
      ix_Activate : Bool;   // Activete statistics counters
      ix_RTrigActivate : Bool;   // Activation rise trigger
   END_VAR

   VAR_IN_OUT
      iqUDT_Statistics : "UDT_EventStatistic";   // Statistic structure
   END_VAR


BEGIN
	(*
	----------------------------------------------------------------------------------------

	Version history:
	Date        | Version   | Author        | Remark
	----------------------------------------------------------------------------------------
	24/05/2019  | 0.1       | C. Leite      | first release MHS TIA 15.1
	17/07/2019  | 0.2       | A.Nowak       | Add comments
	24/07/2019  | 2.0       | L.Klar        | 2.0 MHS library release TIA 15.1
	27/08/2019  | 2.1       | M.Kurpiers    | Comments adjusted
	04/11/2019  | 2.2       | L.Klar        | 1 second pulse changed from memory bit to DB variable
	12/11/2019  | 3.0       | P.Majka       | 3.0 MHS library release TIA 15.1
	21/02/2023  | 4.0       | F.Baten       | 4.0 Release TIA 17.5
	*)

	REGION 1 - Number of events

	    IF (#ix_RTrigActivate)      // Event occured
	    THEN

	        // Increment the number of times the event occurred and clear the time of the current or last event
	        #iqUDT_Statistics.NumberOfTimes += 1;
	        #iqUDT_Statistics.LastEventSeconds := 0;

	    END_IF;

	END_REGION

	REGION 2 - Event time

	    // 1 shot every 1 sec and activate statistic counter
	    IF ("DB_Memory".OS_1sec AND #ix_Activate)
	    THEN

	        // Increment the time of the current or last event and the time of all events that occured
	        #iqUDT_Statistics.LastEventSeconds += 1;
	        #iqUDT_Statistics.TotalEventSeconds += 1;

	    END_IF;

	END_REGION

	REGION 3 - Data reset


	    IF (#ix_Reset)                                            // Reset statistics data
	    THEN

	        IF (NOT #ix_Activate)                                 // Statistic counter isn't activate
	        THEN

	            // Clear statistics data
	            #iqUDT_Statistics.NumberOfTimes := 0;
	            #iqUDT_Statistics.LastEventSeconds := 0;
	            #iqUDT_Statistics.TotalEventSeconds := 0;

	        ELSE

	            // Write 1 to the number of times the event occurred and clear times
	            #iqUDT_Statistics.NumberOfTimes := 1;
	            #iqUDT_Statistics.LastEventSeconds := 0;
	            #iqUDT_Statistics.TotalEventSeconds := 0;

	        END_IF;

	    END_IF;

	END_REGION
END_FUNCTION

FUNCTION_BLOCK "FB_TimerOnOffDelay"
TITLE = FB_TimerOnOffDelay
{ S7_Optimized_Access := 'TRUE' }
AUTHOR : MHSE
FAMILY : GeneralSystemFunctions
VERSION : 3.0
// ATTRIBUTES
// AUTO_NUMBER = True
// BLOCK_NUMBER = 32
// END_ATTRIBUTES
//Function block to generate on/off signal delay.
   VAR_INPUT
      iudi_OnDelayTime { ExternalAccessible := 'False'; ExternalVisible := 'False'; ExternalWritable := 'False'} : UDInt;   // On delay time [ms]
      iudi_OffDelayTime { ExternalAccessible := 'False'; ExternalVisible := 'False'; ExternalWritable := 'False'} : UDInt;   // Off delay time [ms]
      ix_SignalToDelay { ExternalAccessible := 'False'; ExternalVisible := 'False'; ExternalWritable := 'False'} : Bool;   // Input signal to be delayed
      ix_Enable { ExternalAccessible := 'False'; ExternalVisible := 'False'; ExternalWritable := 'False'} : Bool := TRUE;   // Timer Enable
   END_VAR

   VAR_OUTPUT
      qlr_ActualTime { ExternalAccessible := 'False'; ExternalVisible := 'False'; ExternalWritable := 'False'} : LReal;   // Actual time
      qx_DelayedSignal { ExternalAccessible := 'False'; ExternalVisible := 'False'; ExternalWritable := 'False'} : Bool;   // Delayed signal output
   END_VAR

   VAR
      s_R_TRIG_Signal {InstructionName := 'R_TRIG'; LibVersion := '1.0'; ExternalAccessible := 'False'; ExternalVisible := 'False'; ExternalWritable := 'False'; S7_SetPoint := 'False'} : R_TRIG;   // Siemens "R_Trig" - to prepare the rising edge trigger on "ix_SignalToDelay" signal
      s_F_TRIG_Signal {InstructionName := 'F_TRIG'; LibVersion := '1.0'; ExternalAccessible := 'False'; ExternalVisible := 'False'; ExternalWritable := 'False'; S7_SetPoint := 'False'} : F_TRIG;   // Siemens "F_Trig" - to prepare the falling edge trigger on "ix_SignalToDelay" signal
   END_VAR
   VAR RETAIN
      slr_ActualDelayTime { ExternalAccessible := 'False'; ExternalVisible := 'False'; ExternalWritable := 'False'} : LReal;   // Actual delay time [ms]
   END_VAR


BEGIN
	(*
	----------------------------------------------------------------------------------------

	Version history:
	Date        | Version   | Author        | Remark
	----------------------------------------------------------------------------------------
	24/05/2019  | 0.1       | L.Klar        | first release MHS TIA 15.1
	24/07/2019  | 2.0       | L.Klar        | 2.0 MHS library release TIA 15.1
	26/08/2019  | 2.1       | M.Kurpiers    | Comments adjusted
	04/11/2019  | 2.2       | L.Klar        | Prevoius cycle scan changed from memory to DB variable
	12/11/2019  | 3.0       | P.Majka       | 3.0 MHS library release TIA 15.1
	21/02/2023  | 4.0       | F.Baten       | 4.0 Release TIA 17.5
	*)

	REGION Step 1 – Input signal edge detection

	    #s_R_TRIG_Signal(CLK := #ix_SignalToDelay);


	    #s_F_TRIG_Signal(CLK := #ix_SignalToDelay);

	END_REGION

	REGION Step 2 – Actual delay time initialization

	    IF (#s_R_TRIG_Signal.Q OR #s_F_TRIG_Signal.Q)           // Input signal changed
	    THEN

	        #slr_ActualDelayTime := 0;

	    END_IF;

	END_REGION

	REGION Step 3 – On/Off delay time calculation


	    IF (#ix_SignalToDelay                                       // Signal to be delayed is active
	        AND #ix_Enable)                                         // Ttimer enabled
	    THEN

	        // Timer on
	        IF (#slr_ActualDelayTime >= #iudi_OnDelayTime)
	        THEN

	            #qx_DelayedSignal := TRUE;

	        ELSE

	            #slr_ActualDelayTime += "DB_Memory".PrevCycleTime;

	        END_IF;

	    END_IF;

	    // Timer off
	    IF (NOT #ix_SignalToDelay                                   // Signal to delay is not active
	        AND #ix_Enable)                                         // Timer is enabled
	    THEN

	        IF (#slr_ActualDelayTime >= #iudi_OffDelayTime)
	        THEN

	            #qx_DelayedSignal := FALSE;

	        ELSE

	            #slr_ActualDelayTime += "DB_Memory".PrevCycleTime;

	        END_IF;

	    END_IF;

	END_REGION

	REGION Step 4 – Actual time

	    #qlr_ActualTime := #slr_ActualDelayTime;

	END_REGION
END_FUNCTION_BLOCK

TYPE "UDT_TCPIPConnectStatus"
TITLE = UDT_TCPIPConnectStatus
VERSION : 0.1
//User-defined structure of FB_TCPIPConnect function block status.
   STRUCT
      Status : Int;   // Status number
      Specific : Struct   // Specific status structure
         ErrorCode : Struct   // Error code structure
            TCON : Word;   // Siemens TCON error code - Check documetation
            TDISCON : Word;   // Siemens TDISCON error code - Check documetation
            TDIAG : Word;   // Siemens TDIAG error code - Check documetation
         END_STRUCT;
         Connected { ExternalAccessible := 'False'; ExternalVisible := 'False'; ExternalWritable := 'False'} : Bool;   // Connected
         CommunicationFault { ExternalAccessible := 'False'; ExternalVisible := 'False'; ExternalWritable := 'False'} : Bool;   // Communication fault
      END_STRUCT;
   END_STRUCT;

END_TYPE

FUNCTION "FC_Fifo" : Void
TITLE = FC_Fifo
{ S7_Optimized_Access := 'TRUE' }
AUTHOR : MHSE
FAMILY : GeneralSystemFunctions
VERSION : 3.0
// ATTRIBUTES
// AUTO_NUMBER = True
// BLOCK_NUMBER = 17
// END_ATTRIBUTES
//Function for controlling FIFO register.
   VAR_INPUT
      ic_Mode : Char;   // Mode selector: "W" - Write; "R" - Read; "C" - Clear (Reset) "S" - Status
   END_VAR

   VAR_OUTPUT
      qUDT_Status : "UDT_FifoStatus";   // FIFO status structure
      qx_Error : Bool;   // Collective error output
      qx_Warning : Bool;   // Collective warning output
   END_VAR

   VAR_IN_OUT
      iqv_Data : Variant;   // Data
      iqUDT_FifoHeader : "UDT_FifoHeader";   // FIFO header
      iqv_DataBuffer : Variant;   // FIFO data buffer
   END_VAR

   VAR_TEMP
      tUDT_Status : "UDT_FifoStatus";   // Status structure
      ti_MoveBLKErrorCode : Int;   // Move_BLK_Variant function return
      tx_HeaderValid : Bool;   // Header valid
   END_VAR


BEGIN
	(*
	----------------------------------------------------------------------------------------

	Version history:
	Date        | Version   | Author        | Remark
	----------------------------------------------------------------------------------------
	24/05/2019  | 0.1       | L.Klar        | first release MHS TIA 15.1
	14/06/2019  | 0.2       | A.Nowak       | Replacement of instruction if for direct write into variable - Region 3 , 4.1 , 4.2 , 4.3 , 4.4 , 8.1  , 8.2
	17/07/2019  | 0.3       | L.Klar        | Status handling changed
	24/07/2019  | 2.0       | L.Klar        | 2.0 MHS library release TIA 15.1
	23/08/2019  | 2.1       | K.Pokorski    | Comments corrected
	27/08/2019  | 2.2       | M.Kurpiers    | Comments adjusted
	27/09/2019  | 2.3       | K.Pokorski    | Variant input included
	01/10/2019  | 2.4       | A.Nowak       | Correct comments and rename regions
	12/11/2019  | 3.0       | P.Majka       | 3.0 MHS library release TIA 15.1
	21/02/2023  | 4.0       | F.Baten       | 4.0 Release TIA 17.5
	*)

	REGION 1 – Diagnostic bits initialization

	    // Clear FIFO statuses
	    #tUDT_Status.FifoFull := FALSE;
	    #tUDT_Status.FifoPreFull := FALSE;

	END_REGION

	REGION 2 – Array's information

	    // If buffer elements type is invalid, set the error
	    #tUDT_Status.InvalidDataType := NOT (TypeOf(#iqv_Data) = TypeOfElements(#iqv_DataBuffer));

	END_REGION

	REGION 3 – Mode validation

	    // Set the mode invalid if selected mode isn't one of the following: W- Write, R - Read, C - Clear, S - Status
	    #tUDT_Status.InvalidMode := #ic_Mode <> 'W'
	    AND #ic_Mode <> 'R'
	    AND #ic_Mode <> 'C'
	    AND #ic_Mode <> 'S';

	END_REGION

	REGION 4 – The header settings checking

	    // The correct mode has been selected and data type is valid
	    IF (NOT #tUDT_Status.InvalidMode
	        AND NOT #tUDT_Status.InvalidDataType)
	    THEN

	        REGION 4.1 – The number of maximum FIFO entries validation

	            // Write the number of array's elements to FIFO header
	            #iqUDT_FifoHeader.MaxNrOfEntries := "FC_GetNrOfArrayEl"(#iqv_DataBuffer);

	            // Set the invalid maximum number of entries error
	            #tUDT_Status.InvalidMaxNrOfEntries := #iqUDT_FifoHeader.MaxNrOfEntries <= 0;

	        END_REGION

	        REGION 4.2 – The number of total FIFO entries validation

	            // Set the invalid total number of entries error
	            #tUDT_Status.InvalidTotalEntriesStored := #iqUDT_FifoHeader.TotalEntriesStored < 0        // The total number of entries is lower than 0
	            OR #iqUDT_FifoHeader.TotalEntriesStored > #iqUDT_FifoHeader.MaxNrOfEntries;               // The total number of entries is greater than the maximum number of entries

	        END_REGION

	        REGION 4.3 – The number of the next entry to write

	            // Set the invalid next entry to write
	            #tUDT_Status.InvalidNextEntryToWrite := #iqUDT_FifoHeader.NextEntryToWrite < 0            // The number of next entry to write is lower than 0
	            OR #iqUDT_FifoHeader.NextEntryToWrite >= #iqUDT_FifoHeader.MaxNrOfEntries;                // The number of next entry to write is greater or equal to the maximum number of entries

	        END_REGION

	        REGION 4.4 – The number of the next entry to read

	            // Set the invalid next entry to read
	            #tUDT_Status.InvalidNextEntryToRead := #iqUDT_FifoHeader.NextEntryToRead < 0              // The number of next entry to read is lower than 0
	            OR #iqUDT_FifoHeader.NextEntryToRead >= #iqUDT_FifoHeader.MaxNrOfEntries;                 // The number of next entry to read is greater or equal to the maximum nr of entries

	        END_REGION

	        REGION 4.5 – FIFO header validation summary

	            // Create collective header error
	            #tx_HeaderValid := NOT #tUDT_Status.InvalidMaxNrOfEntries
	            AND NOT #tUDT_Status.InvalidTotalEntriesStored
	            AND NOT #tUDT_Status.InvalidNextEntryToWrite
	            AND NOT #tUDT_Status.InvalidNextEntryToRead;

	        END_REGION

	    END_IF;

	END_REGION

	REGION 5 – Writing the data into the FIFO buffer

	    IF (#ic_Mode = 'W'                                                                          // Write mode selected
	        AND #tx_HeaderValid                                                                     // FIFO header valid
	        AND NOT #tUDT_Status.InvalidDataType)                                                  // Buffer data type valid
	    THEN


	        IF (#iqUDT_FifoHeader.TotalEntriesStored < #iqUDT_FifoHeader.MaxNrOfEntries)          // Checking total number of stored entries
	        THEN

	            // Move input data to FIFO data buffer
	            #ti_MoveBLKErrorCode := MOVE_BLK_VARIANT(SRC := #iqv_Data,
	                                                     COUNT := 1,
	                                                     SRC_INDEX := 0,
	                                                     DEST_INDEX := #iqUDT_FifoHeader.NextEntryToWrite,
	                                                     DEST => #iqv_DataBuffer);

	            // Increment the number of the next entry to write
	            #iqUDT_FifoHeader.NextEntryToWrite += 1;

	            // Increment the total number of stored entries
	            #iqUDT_FifoHeader.TotalEntriesStored += 1;


	            IF (#iqUDT_FifoHeader.NextEntryToWrite >= #iqUDT_FifoHeader.MaxNrOfEntries)       // Check the number of the next entry to write
	            THEN

	                #iqUDT_FifoHeader.NextEntryToWrite := 0;

	            END_IF;

	        ELSE

	            #tUDT_Status.FifoFull := TRUE;

	        END_IF;

	    END_IF;

	END_REGION

	REGION 6 – Reading the data from the FIFO data buffer

	    IF (#ic_Mode = 'R'                                                                  // Read mode selected
	        AND #tx_HeaderValid                                                             // FIFO header valid
	        AND NOT #tUDT_Status.InvalidDataType)                                           // Buffer data type valid
	    THEN

	        IF (#iqUDT_FifoHeader.TotalEntriesStored > 0)                                   // Checking total number of stored entries
	        THEN

	            // Move the FIFO data to the data output
	            #ti_MoveBLKErrorCode := MOVE_BLK_VARIANT(SRC := #iqv_DataBuffer,
	                                                     COUNT := 1,
	                                                     SRC_INDEX := #iqUDT_FifoHeader.NextEntryToRead,
	                                                     DEST_INDEX := 0,
	                                                     DEST => #iqv_Data);

	            // Increment the number of the next entry to read
	            #iqUDT_FifoHeader.NextEntryToRead += 1;

	            // Decrement the total number of stored entries
	            #iqUDT_FifoHeader.TotalEntriesStored -= 1;

	            IF (#iqUDT_FifoHeader.NextEntryToRead >= #iqUDT_FifoHeader.MaxNrOfEntries)  // Check the number of the next entry to read
	            THEN

	                #iqUDT_FifoHeader.NextEntryToRead := 0;

	            END_IF;

	        END_IF;

	    END_IF;

	END_REGION

	REGION 7 – Clearing the FIFO header

	    IF (#ic_Mode = 'C'                      // Clear mode selected
	        AND #tx_HeaderValid)                // FIFO header valid
	    THEN

	        #iqUDT_FifoHeader.TotalEntriesStored := 0;
	        #iqUDT_FifoHeader.NextEntryToWrite := 0;
	        #iqUDT_FifoHeader.NextEntryToRead := 0;

	    END_IF;

	END_REGION

	REGION 8 – FIFO management status update

	    IF (#tx_HeaderValid)                   // The header is valid
	    THEN

	        REGION 8.1 – FIFO Empty

	            // Set the FIFO empty status bit
	            #iqUDT_FifoHeader.Status.Empty := #iqUDT_FifoHeader.TotalEntriesStored = 0;

	        END_REGION

	        REGION 8.2 – FIFO Full

	            // Set the FIFO full status bit
	            #iqUDT_FifoHeader.Status.Full := #iqUDT_FifoHeader.TotalEntriesStored = #iqUDT_FifoHeader.MaxNrOfEntries;

	        END_REGION

	        REGION 8.3 – FIFO Pre-full

	            IF (#iqUDT_FifoHeader.TotalEntriesStored >= 0.9 * #iqUDT_FifoHeader.MaxNrOfEntries)       // Checking if the number of total stored entries is greater or equal to 90% of the max number of entries
	            THEN

	                // Set the FIFO pre-full status
	                #iqUDT_FifoHeader.Status.Prefull := TRUE;
	                #tUDT_Status.FifoPreFull := TRUE;

	            ELSE

	                #iqUDT_FifoHeader.Status.Prefull := FALSE;

	            END_IF;

	        END_REGION

	    END_IF;

	END_REGION

	REGION 9 – Status

	    REGION 9.1 – Common status update

	        // Collective error output
	        #qx_Error := NOT #tx_HeaderValid
	        OR #tUDT_Status.InvalidMode
	        OR #tUDT_Status.FifoFull
	        OR #tUDT_Status.InvalidDataType;

	        // Collective warning output
	        #qx_Warning := #tUDT_Status.FifoPreFull;

	    END_REGION

	    REGION 9.2 – Status update

	        // Update the outer status structure with internal status structure
	        #qUDT_Status := #tUDT_Status;

	    END_REGION

	END_REGION
END_FUNCTION

TYPE "UDT_TCPIPReceiveStatistics"
TITLE = UDT_TCPIPReceiveStatistics
VERSION : 0.1
//User-defined structure of FB_TCPIPReceive function block statistics.
   STRUCT
      InvalidMsg : UInt;   // Invalid message received
   END_STRUCT;

END_TYPE

FUNCTION_BLOCK "FB_Pulse"
TITLE = FB_Pulse
{ S7_Optimized_Access := 'TRUE' }
AUTHOR : MHSE
FAMILY : GeneralSystemFunctions
VERSION : 3.0
// ATTRIBUTES
// AUTO_NUMBER = True
// BLOCK_NUMBER = 26
// END_ATTRIBUTES
//Function block to generate custom pulse signal.
   VAR_INPUT
      iudi_PulseTime { ExternalAccessible := 'False'; ExternalVisible := 'False'; ExternalWritable := 'False'} : UDInt;   // Pulse time [ms]
   END_VAR

   VAR_OUTPUT
      qx_Pulse { ExternalAccessible := 'False'; ExternalVisible := 'False'; ExternalWritable := 'False'} : Bool;   // Pulse output
   END_VAR

   VAR
      R_TRIG {InstructionName := 'R_TRIG'; LibVersion := '1.0'; ExternalAccessible := 'False'; ExternalVisible := 'False'; ExternalWritable := 'False'; S7_SetPoint := 'False'} : R_TRIG;   // Siemens "R_Trig" - to prepare rising edge trigger on "sx_Pulse" signal
      slr_ActualPulseTime { ExternalAccessible := 'False'; ExternalVisible := 'False'; ExternalWritable := 'False'} : LReal;   // Actual pulse time [ms]
      sx_Pulse { ExternalAccessible := 'False'; ExternalVisible := 'False'; ExternalWritable := 'False'} : Bool;   // Pulse signal
   END_VAR


BEGIN
	(*
	----------------------------------------------------------------------------------------

	Version history:
	Date        | Version   | Author        | Remark
	----------------------------------------------------------------------------------------
	24/05/2019  | 0.1       | K.Pokorski    | first release MHS TIA 15.1
	24/07/2019  | 2.0       | L.Klar        | 2.0 MHS library release TIA 15.1
	27/08/2019  | 2.1       | K.Pokorski    | Comments adjusted
	04/11/2019  | 2.2       | L.Klar        | Prevoius cycle scan changed from memory to DB variable
	12/11/2019  | 3.0       | P.Majka       | 3.0 MHS library release TIA 15.1
	21/02/2023  | 4.0       | F.Baten       | 4.0 Release TIA 17.5
	*)

	REGION 1 - Pulse calculation

	    // Pulse timer on
	    IF (#iudi_PulseTime <= #slr_ActualPulseTime)
	    THEN

	        #sx_Pulse := TRUE;
	        #slr_ActualPulseTime := 0;

	    ELSE

	        #slr_ActualPulseTime += "DB_Memory".PrevCycleTime;
	        #sx_Pulse := FALSE;

	    END_IF;

	END_REGION

	REGION 2 - Pulse output

	    #R_TRIG(CLK := #sx_Pulse,
	            Q => #qx_Pulse);

	END_REGION
END_FUNCTION_BLOCK

TYPE "UDT_UPSHeartbeatStatistics"
TITLE = UDT_HeartbeatStatistics
VERSION : 0.1
//User-defined structure of FB_Heartbeat function block statistics.
   STRUCT
      ConLost : UDInt;   // Statistics of connection lost
   END_STRUCT;

END_TYPE

TYPE "UDT_UPSMSGIDCounters"
VERSION : 0.1
   STRUCT
      Heartbeat : DInt;   // Heartbeat MSGID counter
      IDFWD : DInt;   // IDFWD MSGID counter
      SORTCONF : DInt;   // SORTCONF MSGID counter
      PLCINFO : DInt;   // PLCINFO MSGID counter
      SORT : DInt;   // SORT MSGID counter
      HB : DInt;   // HB MSGID counter
   END_STRUCT;

END_TYPE

TYPE "UDT_UPSDecodeStatistics"
TITLE = UDT_DecodeStatistics
VERSION : 0.1
//User-defined structure of FB_Decode function block statistics.
   STRUCT
      InvalidMsg : UDInt;   // Counter of incorrectly decoded messages
      HBNotObserved : UDInt;   // Statistics of HB not observed in a preset time
   END_STRUCT;

END_TYPE

TYPE "UDT_UPSCIPStatistics"
VERSION : 0.1
   STRUCT
      CIP24VDCFault : "UDT_EventStatistic";   // 24V fault
      CIPCircuitBreakerTripped : "UDT_EventStatistic";   // Circuit breaker tripped
      WeighingScaleFault : "UDT_EventStatistic";   // Weighing scale fault
      SS_Camera { S7_SetPoint := 'True'} : DInt;   // Number of times camera switch change over
      SS_XLE { S7_SetPoint := 'True'} : DInt;   // Number of times XLE switch change over
   END_STRUCT;

END_TYPE

FUNCTION "FC_SeparateMsg" : Void
TITLE = FC_SeparateMsg
{ S7_Optimized_Access := 'TRUE' }
AUTHOR : MHSE
FAMILY : GeneralSystemFunctions
VERSION : 3.0
// ATTRIBUTES
// AUTO_NUMBER = True
// BLOCK_NUMBER = 25
// END_ATTRIBUTES
//Function to separate the delimited message.
   VAR_INPUT
      iUDT_Message : "UDT_Message";   // Character string to be separated
      ii_Position : Int;   // Start position
      ic_Delimiter : Char;   // Delimiter
      ic_EndSign : Char;   // End of the message sign
   END_VAR

   VAR_OUTPUT
      qs_Msg : String;   // Separated part of the message
      qui_Length : UInt;   // Length of the separated message
      qx_EndMsg : Bool;   // End message sign found
      qx_NoSeparationSign : Bool;   // Separation sign not detected
   END_VAR

   VAR_TEMP
      ti_i : Int;   // Loop counter
      tui_NrOfConvChar : UInt;   // Number of converted message characters
      ti_SizeOfMsg : Int;   // Message array size
   END_VAR


BEGIN
	(*
	----------------------------------------------------------------------------------------

	Version history:
	Date        | Version   | Author        | Remark
	----------------------------------------------------------------------------------------
	24/05/2019  | 0.1       | K.Pokorski    | first release MHS TIA 15.1
	14/06/2019  | 0.2       | K.Pokorski    | "ii_Position" input, "qx_NoSeparationSign" output added, additional logic programmed
	17/06/2019  | 0.3       | L.Klar        | "iqi_Position" deleted
	24/07/2019  | 2.0       | L.Klar        | 2.0 MHS library release TIA 15.1
	26/07/2019  | 2.1       | M.Kurpiers    | Comments adjusted
	12/11/2019  | 3.0       | P.Majka       | 3.0 MHS library release TIA 15.1
	21/02/2023  | 4.0       | F.Baten       | 4.0 Release TIA 17.5
	*)

	REGION 1 – Maximum number of the message characters

	    #ti_SizeOfMsg := "FC_GetNrOfArrayEl"(iv_Array := #iUDT_Message.Character);

	END_REGION

	REGION 2 – Message separation

	    IF (#ii_Position <= #ti_SizeOfMsg - 1)                                        // Position is lower than size of a message array
	    THEN

	        // Delimiter and end sign search loop
	        FOR #ti_i := #ii_Position TO #ti_SizeOfMsg - 1 DO


	            IF (#iUDT_Message.Character[#ti_i] = #ic_Delimiter                    // Check if delimiter and the end of the message was found
	                OR #iUDT_Message.Character[#ti_i] = #ic_EndSign)

	            THEN

	                // Message length minus start position from INT to UInt conversion
	                #tui_NrOfConvChar := INT_TO_UINT(IN := (#ti_i - #ii_Position));

	                IF #tui_NrOfConvChar <> 0
	                THEN
	                    // Character array into the message character string conversion
	                    Chars_TO_Strg(Chars := #iUDT_Message.Character,
	                                  pChars := #ii_Position,
	                                  Cnt := #tui_NrOfConvChar,
	                                  Strg => #qs_Msg);

	                ELSE
	                    #qs_Msg := '';
	                END_IF;

	                // Length of the separated message part
	                #qui_Length := #tui_NrOfConvChar;

	                // Separation sign not detected
	                #qx_NoSeparationSign := FALSE;


	                IF (#iUDT_Message.Character[#ti_i] = #ic_EndSign)                   // End of the message sign detected
	                THEN

	                    #qx_EndMsg := TRUE;

	                ELSE

	                    #qx_EndMsg := FALSE;

	                END_IF;
	                // Exit the loop if end sign was found
	                EXIT;


	            ELSIF (#ti_i = #ti_SizeOfMsg - 1)                                         // Separate sign is not detected
	            THEN

	                // End of the message and no separation sign detected bits are set
	                #qs_Msg := '';
	                #qui_Length := 0;
	                #qx_EndMsg := TRUE;
	                #qx_NoSeparationSign := TRUE;

	            END_IF;

	        END_FOR;
	        // Clear variables if delimiter and end sign wasn't found
	    ELSE

	        #qs_Msg := '';
	        #qui_Length := 0;
	        #qx_EndMsg := TRUE;
	        #qx_NoSeparationSign := TRUE;

	    END_IF;

	END_REGION
END_FUNCTION

TYPE "UDT_UPSFlowControlHMI"
VERSION : 0.1
   STRUCT
      Setpoint : Int;   // Setpoint value from HMI
      CalculatedFlow : Int;   // Current calculated value to HMI
      CommandToDisable : Bool;   // Command from HMI to disable
      DisabledStatus : Bool;   // Disabled Status
   END_STRUCT;

END_TYPE

TYPE "UDT_UPSFlowRateCountingRegisters"
VERSION : 0.1
   STRUCT
      iCR : Array[1..60] of Int;   // Counting Register
   END_STRUCT;

END_TYPE

FUNCTION "FC_UPSScanData2" : Void
TITLE = FC_Health
{ S7_Optimized_Access := 'TRUE' }
AUTHOR : MHSE
FAMILY : UPS_SpecificCommunication
VERSION : 3.0
// ATTRIBUTES
// AUTO_NUMBER = True
// BLOCK_NUMBER = 35
// END_ATTRIBUTES
//Function to decode the UPS HEALTH message.
   VAR_INPUT
      iUDT_Message : "UDT_UPSMessage";   // Sorted message
   END_VAR

   VAR_OUTPUT
      qx_Error : Bool;   // Error
   END_VAR

   VAR_IN_OUT
      iqa_ExternalReaders : Array[*] of "UDT_UPSExternalReader";   // Health structure
   END_VAR

   VAR_TEMP
      ti_i : Int;   // Loop counter
      ti_j : Int;   // Loop counter
      ti_ExternalReadersArrayLength : Int;   // External readers array length
      ti_ExternalReadersArrayLowBound : Int;   // External readers array low bound
      tusi_PackageNr : Int;
   END_VAR


BEGIN
	(*
	----------------------------------------------------------------------------------------

	Version history:
	Date        | Version   | Author        | Remark
	----------------------------------------------------------------------------------------
	24/05/2019  | 0.1       | K.Pokorski    | first release MHS TIA 15.1
	14/06/2019  | 0.2       | A.Nowak       | Replacement of instruction if for direct write into variable - Region 3
	24/07/2019  | 2.0       | L.Klar        | 2.0 MHS library release TIA 15.1
	23/08/2019  | 2.1       | K.Pokorski    | Comments simplified
	12/11/2019  | 3.0       | P.Majka       | 3.0 MHS library release TIA 15.1
	01/07/2020  | 3.1       | L.Klar        | Block changed to fit new SCAN DATA 2 message template
	14/12/2020  | 3.2       | L.Klar        | ID created bit added
	21/02/2023  | 4.0       | F.Baten       | 4.0 Release TIA 17.5
	*)

	REGION 1 – Initialization

	    #ti_ExternalReadersArrayLength := "FC_GetNrOfArrayEl"(#iqa_ExternalReaders);
	    #ti_ExternalReadersArrayLowBound := DINT_TO_INT(LOWER_BOUND(ARR := #iqa_ExternalReaders, DIM := 1));

	END_REGION

	REGION 2 – Message handling

	    // Loop used to find message sender (external reader) in configured array
	    FOR #ti_i := #ti_ExternalReadersArrayLowBound TO #ti_ExternalReadersArrayLowBound + #ti_ExternalReadersArrayLength - 1 DO

	        IF (#iUDT_Message.SCT = #iqa_ExternalReaders[#ti_i].NameIdentifier)
	        THEN

	            #iqa_ExternalReaders[#ti_i].ScanData2Message.MSGID := #iUDT_Message.Data[1];
	            #iqa_ExternalReaders[#ti_i].ScanData2Message.CONFLICT_CODE := #iUDT_Message.Data[2];
	            #iqa_ExternalReaders[#ti_i].ScanData2Message.BARCODE_ZIP := #iUDT_Message.Data[3];
	            #iqa_ExternalReaders[#ti_i].ScanData2Message.BARCODE_TRACK := #iUDT_Message.Data[4];
	            #iqa_ExternalReaders[#ti_i].ScanData2Message.BARCODE_PTN := #iUDT_Message.Data[5];
	            #iqa_ExternalReaders[#ti_i].ScanData2Message.MAXI_ZIPCODE := #iUDT_Message.Data[6];
	            #iqa_ExternalReaders[#ti_i].ScanData2Message.MAXI_COUNTRY := #iUDT_Message.Data[7];
	            #iqa_ExternalReaders[#ti_i].ScanData2Message.MAXI_SERVICE := #iUDT_Message.Data[8];
	            #iqa_ExternalReaders[#ti_i].ScanData2Message.MAXI_TRACK := #iUDT_Message.Data[9];
	            #iqa_ExternalReaders[#ti_i].ScanData2Message.MAXI_SHIPPER := #iUDT_Message.Data[10];
	            #iqa_ExternalReaders[#ti_i].ScanData2Message.LENGTH1 := #iUDT_Message.Data[11];
	            #iqa_ExternalReaders[#ti_i].ScanData2Message.LENGTH2 := #iUDT_Message.Data[12];
	            #iqa_ExternalReaders[#ti_i].ScanData2Message.HEIGHT := #iUDT_Message.Data[13];
	            #iqa_ExternalReaders[#ti_i].ScanData2Message.VERTEX := #iUDT_Message.Data[14];
	            #iqa_ExternalReaders[#ti_i].ScanData2Message.ORIENTATION := #iUDT_Message.Data[15];
	            #iqa_ExternalReaders[#ti_i].ScanData2Message.OVERHANG := #iUDT_Message.Data[16];
	            #iqa_ExternalReaders[#ti_i].ScanData2Message.WEIGHT := #iUDT_Message.Data[17];
	            #iqa_ExternalReaders[#ti_i].ScanData2Message.APPENDED_DATA.Constant_1 := #iUDT_Message.Data[18];
	            #iqa_ExternalReaders[#ti_i].ScanData2Message.APPENDED_DATA.FRAME_ID := #iUDT_Message.Data[19];
	            #iqa_ExternalReaders[#ti_i].ScanData2Message.APPENDED_DATA.DIMENSION := #iUDT_Message.Data[20];
	            #iqa_ExternalReaders[#ti_i].ScanData2Message.APPENDED_DATA.PACKAGE_NUMBER := #iUDT_Message.Data[21];
	            #iqa_ExternalReaders[#ti_i].ScanData2Message.APPENDED_DATA.BARCODE_1 := #iUDT_Message.Data[22];
	            #iqa_ExternalReaders[#ti_i].ScanData2Message.APPENDED_DATA.DESCRIPTION_1 := #iUDT_Message.Data[23];
	            #iqa_ExternalReaders[#ti_i].ScanData2Message.APPENDED_DATA.BARCODE_2 := #iUDT_Message.Data[24];
	            #iqa_ExternalReaders[#ti_i].ScanData2Message.APPENDED_DATA.DESCRIPTION_2 := #iUDT_Message.Data[25];
	            #iqa_ExternalReaders[#ti_i].ScanData2Message.APPENDED_DATA.BARCODE_3 := #iUDT_Message.Data[26];
	            #iqa_ExternalReaders[#ti_i].ScanData2Message.APPENDED_DATA.DESCRIPTION_3 := #iUDT_Message.Data[27];
	            #iqa_ExternalReaders[#ti_i].ScanData2Message.APPENDED_DATA.Constant_4 := #iUDT_Message.Data[28];
	            #iqa_ExternalReaders[#ti_i].ScanData2Message.APPENDED_DATA.SCALE_WEIGHT := #iUDT_Message.Data[29];
	            #iqa_ExternalReaders[#ti_i].ScanData2Message.APPENDED_DATA.Constant_5 := #iUDT_Message.Data[30];
	            #iqa_ExternalReaders[#ti_i].ScanData2Message.APPENDED_DATA.GIRTH := #iUDT_Message.Data[31];
	            #iqa_ExternalReaders[#ti_i].ScanData2Message.APPENDED_DATA.Constant_6 := #iUDT_Message.Data[32];
	            #iqa_ExternalReaders[#ti_i].ScanData2Message.APPENDED_DATA.ERROR_CODE := #iUDT_Message.Data[33];

	            FOR #ti_j := 1 TO 32 DO

	                IF #iUDT_Message.Data[#ti_j] = '1' THEN

	                    #tusi_PackageNr := STRING_TO_INT(MID(IN := #iUDT_Message.Data[#ti_j + 1], L := 4, P := 3));


	                    IF #tusi_PackageNr > 0 AND #tusi_PackageNr < 9999
	                    THEN
	                        "DB_GIN".GIN[#tusi_PackageNr].UPS.IDCreated := TRUE;
	                    END_IF;
	                    EXIT;

	                END_IF;
	            END_FOR;

	            #qx_Error := FALSE;
	            EXIT;

	        ELSE
	            #qx_Error := TRUE;
	        END_IF;
	    END_FOR;

	END_REGION
END_FUNCTION

FUNCTION "FC_UPSHealth" : Void
TITLE = FC_Health
{ S7_Optimized_Access := 'TRUE' }
AUTHOR : MHSE
FAMILY : UPS_SpecificCommunication
VERSION : 3.0
// ATTRIBUTES
// AUTO_NUMBER = True
// BLOCK_NUMBER = 33
// END_ATTRIBUTES
//Function to decode the UPS HEALTH message.
   VAR_INPUT
      iUDT_Message : "UDT_UPSMessage";   // Sorted message
   END_VAR

   VAR_OUTPUT
      qx_Error : Bool;   // Error
   END_VAR

   VAR_IN_OUT
      iqa_ExternalReaders : Array[*] of "UDT_UPSExternalReader";   // Health structure
   END_VAR

   VAR_TEMP
      ti_Failure : DInt;   // External reader failure mask
      ti_i : Int;   // Loop counter
      ti_ExternalReadersArrayLength : Int;   // External readers array length
      ti_ExternalReadersArrayLowBound : Int;   // External readers array low bound
   END_VAR

   VAR CONSTANT
      cs_CAM : String := 'CAM';   // Camera
      cs_DWS : String := 'DWS';   // Scale
   END_VAR


BEGIN
	(*
	----------------------------------------------------------------------------------------

	Version history:
	Date        | Version   | Author        | Remark
	----------------------------------------------------------------------------------------
	24/05/2019  | 0.1       | K.Pokorski    | first release MHS TIA 15.1
	14/06/2019  | 0.2       | A.Nowak       | Replacement of instruction if for direct write into variable - Region 3
	24/07/2019  | 2.0       | L.Klar        | 2.0 MHS library release TIA 15.1
	23/08/2019  | 2.1       | K.Pokorski    | Comments simplified
	12/11/2019  | 3.0       | P.Majka       | 3.0 MHS library release TIA 15.1
	01/07/2020  | 3.1       | L.Klar        | Block changed to fit new HEALHT message template
	22/02/2023  | 4.0       | F.Baten       | 4.0 Release TIA 17.5
	*)

	REGION 1 – Initialization

	    #ti_Failure := 0;

	    #ti_ExternalReadersArrayLength := "FC_GetNrOfArrayEl"(#iqa_ExternalReaders);
	    #ti_ExternalReadersArrayLowBound := DINT_TO_INT(LOWER_BOUND(ARR := #iqa_ExternalReaders, DIM := 1));
	END_REGION

	REGION 2 – Message handling

	    // Loop used to find message sender (external reader) in configured array
	    FOR #ti_i := #ti_ExternalReadersArrayLowBound TO #ti_ExternalReadersArrayLowBound + #ti_ExternalReadersArrayLength - 1 DO

	        IF (#iUDT_Message.SCT = #iqa_ExternalReaders[#ti_i].NameIdentifier)
	        THEN

	            // Device type
	            IF #iUDT_Message.Data[4] = '1'
	            THEN
	                #iqa_ExternalReaders[#ti_i].HealthMessage.Type := #cs_DWS;
	            ELSIF #iUDT_Message.Data[4] = '2'
	            THEN
	                #iqa_ExternalReaders[#ti_i].HealthMessage.Type := #cs_CAM;
	            END_IF;

	            // Device failure mask
	            STRG_VAL(IN := #iUDT_Message.Data[5],
	                     FORMAT := 16#0,
	                     P := 1,
	                     OUT => #ti_Failure);

	            #iqa_ExternalReaders[#ti_i].HealthMessage.Failure := #ti_Failure;

	            // Device model
	            #iqa_ExternalReaders[#ti_i].HealthMessage.Model := #iUDT_Message.Data[6];

	            // Device error
	            #iqa_ExternalReaders[#ti_i].HealthMessage.Error := #ti_Failure > 0;
	            #qx_Error := FALSE;
	            EXIT;

	        ELSE
	            #qx_Error := TRUE;
	        END_IF;
	    END_FOR;

	END_REGION
END_FUNCTION

TYPE "UDT_UPSCIPStatus"
VERSION : 0.1
   STRUCT
      Status : Int;   // Status number
      Specific : Struct
         CIP24VDCError : Bool;   // CIP 24VDC error
         CIPCircuitBreakerTripped : Bool;   // CIP Circuit Breaker Tripped
         XLE_SwitchError : Bool;   // XLE switched while stystem was ruuning
         Camera_SwitchError : Bool;   // Camera switched while stystem was ruuning
         WeighingScaleFault : Bool;   // Weighing Scale Fault
         CameraTunel1 : Bool;   // Camera Tunel 1 Selected
         CameraTunel2 : Bool;   // Camera Tunel 2 Selected
         XLEBackUp : Bool;   // XLE BackUp selected
         XLEPrimary : Bool;   // XLE Primary selected
      END_STRUCT;
   END_STRUCT;

END_TYPE

FUNCTION_BLOCK "FB_UPSAcknowledge"
TITLE = FB_Acknowledge
{ S7_Optimized_Access := 'TRUE' }
AUTHOR : MHSE
FAMILY : UPS_SpecificCommunication
VERSION : 3.0
// ATTRIBUTES
// AUTO_NUMBER = True
// BLOCK_NUMBER = 48
// END_ATTRIBUTES
//Function block to prepare and send the UPS Acknowledge message.
   VAR_INPUT
      iUDT_Message { ExternalAccessible := 'False'; ExternalVisible := 'False'; ExternalWritable := 'False'} : "UDT_UPSMessage";   // Message structure
   END_VAR

   VAR_OUTPUT
      qx_Error { ExternalAccessible := 'False'; ExternalVisible := 'False'; ExternalWritable := 'False'} : Bool;   // Collective error output
      qx_Warning { ExternalAccessible := 'False'; ExternalVisible := 'False'; ExternalWritable := 'False'} : Bool;   // Collective warning output
   END_VAR

   VAR_IN_OUT
      iqUDT_FifoHeader : "UDT_FifoHeader";   // FIFO header
      iqa_FifoData : Array[*] of "UDT_Message";   // FIFO data
   END_VAR

   VAR
      ss_MT { ExternalAccessible := 'False'; ExternalVisible := 'False'; ExternalWritable := 'False'} : String[20];   // Message type character string
      ss_Message { ExternalAccessible := 'False'; ExternalVisible := 'False'; ExternalWritable := 'False'} : String;   // Message character string
      s_UDT_MessageArray { ExternalAccessible := 'False'; ExternalVisible := 'False'; ExternalWritable := 'False'; S7_SetPoint := 'False'} : "UDT_Message";   // Message character array
      sa_Status { ExternalAccessible := 'False'; ExternalVisible := 'False'; ExternalWritable := 'False'} : Struct   // Status structure
         FIFOStatus { ExternalAccessible := 'False'; ExternalVisible := 'False'; ExternalWritable := 'False'} : "UDT_FifoStatus";
         FIFOError { ExternalAccessible := 'False'; ExternalVisible := 'False'; ExternalWritable := 'False'; S7_SetPoint := 'True'} : Bool;   //   FIFO error
         FIFOWarning { ExternalAccessible := 'False'; ExternalVisible := 'False'; ExternalWritable := 'False'; S7_SetPoint := 'True'} : Bool;   //   FIFO warning
      END_STRUCT;
      sui_ArrayOffset { ExternalAccessible := 'False'; ExternalVisible := 'False'; ExternalWritable := 'False'} : UInt;   // Offset for writing in the array
      si_MaxMsgLen { ExternalAccessible := 'False'; ExternalVisible := 'False'; ExternalWritable := 'False'} : Int;   // Maximum message length
   END_VAR

   VAR CONSTANT
      cs_ACK : String := 'ACK-';   // Message type
      cs_CRLF : String := '$R$L';   // Termination signs
      cc_DL : Char := ',';   // Comma sign
   END_VAR


BEGIN
	(*
	----------------------------------------------------------------------------------------

	Version history:
	Date        | Version   | Author        | Remark
	----------------------------------------------------------------------------------------
	24/05/2019  | 0.1       | L.Klar        | first release MHS TIA 15.1
	28/06/2019  | 0.4       | A.Nowak       | Changing conditions for error occuring and status update
	17/07/2019  | 0.5       | L.Klar        | Status handling changed
	24/07/2019  | 2.0       | L.Klar        | 2.0 MHS library release TIA 15.1
	23/08/2019  | 2.1       | K.Pokorski    | Comments simplified
	20/09/2019  | 2.2       | A.Nowak       | Change data type of Status from "UDT_Status" to Struct
	01/10/2019  | 2.3       | A.Nowak       | Implementation of the new FIFO block
	12/11/2019  | 3.0       | P.Majka       | 3.0 MHS library release TIA 15.1
	22/02/2023  | 4.0       | F.Baten       | 4.0 Release TIA 17.5
	*)

	REGION 1 – Update FIFO header status bits

	    // Mode 'S' - FIFO register status update
	    "FC_Fifo"(ic_Mode := 'S',
	              qUDT_Status => #sa_Status.FIFOStatus,
	              qx_Error => #sa_Status.FIFOError,
	              qx_Warning => #sa_Status.FIFOWarning,
	              iqv_Data := #s_UDT_MessageArray,
	              iqUDT_FifoHeader := #iqUDT_FifoHeader,
	              iqv_DataBuffer := #iqa_FifoData);

	END_REGION

	REGION 2 – ACK message preparation

	    IF (NOT #sa_Status.FIFOError)                            // No FIFO error
	    THEN

	        IF (NOT #iqUDT_FifoHeader.Status.Full)                 // FIFO not full
	        THEN

	            REGION 2.1 – Message type preparation

	                // Add "ACK-" prefix into the original messege type
	                #ss_MT := CONCAT(IN1 := #cs_ACK, IN2 := #iUDT_Message.MT);

	            END_REGION

	            REGION 2.2 – Message preparation

	                // Acknowledge message composing according to the structure: SCN,SCT,RCN,RCT,MT+'ACK',MSGID {CRLF}
	                #ss_Message := CONCAT(IN1 := #iUDT_Message.RCN,            // Receiver IP address ("i_UDT_Message.RCN")
	                                      IN2 := #cc_DL,                        // Comma sign ("cc_DL") - ","
	                                      IN3 := #iUDT_Message.RCT,            // Receiver Name ("i_UDT_Message.RCT")
	                                      IN4 := #cc_DL,                        // Comma sign ("cc_DL") - ","
	                                      IN5 := #iUDT_Message.SCN,            // Sender IP address ("i_UDT_Message.SCN")
	                                      IN6 := #cc_DL,                        // Comma sign ("cc_DL") - ","
	                                      IN7 := #iUDT_Message.SCT,            // Sender Name ("i_UDT_Message.SCT")
	                                      IN8 := #cc_DL,                        // Comma sign ("cc_DL") - ","
	                                      IN9 := #ss_MT,                        // Message type("ss_MT") - "ACK-" + original message type
	                                      IN10 := #cc_DL,                       // Comma sign ("cc_DL") - ","
	                                      IN11 := #iUDT_Message.Data[1],       // Message ID - MSGID ("i_UDT_Message.Data[1]")
	                                      IN12 := #cs_CRLF);                    // Termination signs ("cs_CRLF") - "$R$L"

	            END_REGION

	            REGION 2.3 – Maximum number of message array elements

	                #si_MaxMsgLen := "FC_GetNrOfArrayEl"(iv_Array := #s_UDT_MessageArray.Character);

	            END_REGION

	            REGION 2.4 – Message character string conversion to a message array of characters

	                Strg_TO_Chars(Strg := #ss_Message,
	                              pChars := 0,
	                              Cnt => #sui_ArrayOffset,
	                              Chars := #s_UDT_MessageArray.Character);

	            END_REGION

	            REGION 2.5 – Clearing remaining characters in the message character array

	                // Filling up not used message character array elements with '$00' (ASCII - 16#00)
	                FILL_BLK(IN := '$00',
	                         COUNT := UINT_TO_ULINT(INT_TO_UINT(#si_MaxMsgLen) -
	                                                #sui_ArrayOffset),
	                         OUT => #s_UDT_MessageArray.Character[#sui_ArrayOffset]);

	            END_REGION

	            REGION 2.6 – Message write into a FIFO register

	                // Mode 'W' - Write FIFO record
	                "FC_Fifo"(ic_Mode := 'W',
	                          qUDT_Status => #sa_Status.FIFOStatus,
	                          qx_Error => #sa_Status.FIFOError,
	                          qx_Warning => #sa_Status.FIFOWarning,
	                          iqv_Data := #s_UDT_MessageArray,
	                          iqUDT_FifoHeader := #iqUDT_FifoHeader,
	                          iqv_DataBuffer := #iqa_FifoData);

	            END_REGION

	            // In case of FIFO full, the FIFO full error bit and FIFO collective error bit are set
	        ELSE

	            #sa_Status.FIFOError := TRUE;
	            #sa_Status.FIFOStatus.FifoFull := TRUE;

	        END_IF;

	    END_IF;

	END_REGION

	REGION 3 – Status

	    // Parametrization collective error output
	    #qx_Error := #sa_Status.FIFOError;           // FIFO error

	    // Parametrization collective warning output
	    #qx_Warning := #sa_Status.FIFOWarning;       // FIFO warning

	END_REGION
END_FUNCTION_BLOCK

TYPE "UDT_UPSChatStatistics"
VERSION : 0.1
   STRUCT
      CommunicationError : "UDT_EventStatistic";
      LostChatConnection : "UDT_EventStatistic";
      LostXLeConnection : "UDT_EventStatistic";
      LostPLCCommunication : "UDT_EventStatistic";
      Heartbeat { ExternalAccessible := 'False'; ExternalVisible := 'False'; ExternalWritable := 'False'} : DInt;   // Heartbeat message counter
      IDFWD { ExternalAccessible := 'False'; ExternalVisible := 'False'; ExternalWritable := 'False'} : DInt;   // IDFWD message counter
      SORTCONF { ExternalAccessible := 'False'; ExternalVisible := 'False'; ExternalWritable := 'False'} : DInt;   // SORTCONF message counter
      PLCMsg { ExternalAccessible := 'False'; ExternalVisible := 'False'; ExternalWritable := 'False'} : DInt;   // PLCMsg message counter
      PLCINFO { ExternalAccessible := 'False'; ExternalVisible := 'False'; ExternalWritable := 'False'} : DInt;   // PLCINFO message counter
      SORT { ExternalAccessible := 'False'; ExternalVisible := 'False'; ExternalWritable := 'False'} : DInt;   // SORT message counter
      HB : DInt;   // HB message counter
   END_STRUCT;

END_TYPE

TYPE "UDT_UPSMessageHeader"
TITLE = UDT_UPSMessageHeader
VERSION : 0.1
//User-defined structure of UPS message header data.
   STRUCT
      SCN : String[15] := 'aaa.bbb.ccc.ddd';   // Sender client name
      SCT : String[8] := 'AAA-BBBB';   // Sender client type
      RCN : String[15] := 'aaa.bbb.ccc.ddd';   // Receiver client name
      RCT : String[8] := 'AAA-BBBB';   // Receiver client type
   END_STRUCT;

END_TYPE

TYPE "UDT_UPSSspStatistics"
VERSION : 0.1
   STRUCT
      CS_Start : DInt;   // Number of times started
      CS_Stop : "UDT_EventStatistic";
   END_STRUCT;

END_TYPE

